KUKA KRL program: chk_w3_grp3_clo.src

&ACCESS RVO1
&COMMENT Check GRP Z3 ACTROS CLOSE
DEF chk_w3_grp3_clo( )

; Check gripper actros CLOSE Z3
;//---- Start User-------

$TIMER[10] = 0
$TIMER_STOP[10] = FALSE

WAIT FOR (NOT $IN[11])
WAIT FOR ($IN[12])

$TIMER_STOP[10] = TRUE
$TIMER[10] = 0

;//---- End User---------

END
